Yaskawa INFORM job: AAA.JBI

/JOB
//NAME AAA
//POS
///NPOS 1,0,0,0,0,0
///TOOL 9
///POSTYPE PULSE
///PULSE
C00000=-877,2097,1409,61,-956,-71
//INST
///DATE 2023/01/22 23:28
///COMM Generated using RoboDK
///ATTR SC,RW
///GROUP1 RB1
NOP
MOVJ C00000 VJ=1.0 PL=0
END
